(* CODESYS project Initial_Program_RECOVERED_2024-04-08T14-02-49.project
   Version: 0.0.0.0
   Title: Initial_Program
   Author: MYBOOK

Project tree, tasks and I/O mapping:
  Skripsi_Yosef : TM262L10MESE8T, Schneider Electric, order no. TM262L10MESE8T, version 5.0.4.83
      settings: Enable OPC-UA Server = True; BinaryFileSize = 968; Dhcps Host 0.Client Device Name = 'DEVICE_1'; Dhcps Host 0.Client IP Address = [192, 168, 3, 3]; Dhcps Host 0.Network Mask = [255, 255, 255, 0]; Dhcps Host 0.Default Gateway = [192, 168, 3, 254]; serialized Values = 512f82cd-0d03-416a-ab18-865b7c93dff8=0|; InterfaceUsedByDhcpSize = 4; InterfaceUsedByDhcp = [192,168,3,254]
    application Application
      task MAST (cyclic, interval 10 ms, priority 15, watchdog 50 ms x 1) calls SR_Main
      program SR_Main [LD]
      global variables GVL
    Machine Assistant
    Message Logger
    Ethernet_1 : ETH1, Schneider Electric, version 5.0.4.83
        settings: DeviceName = 'M262'; WebServer = FALSE; FTP Server = TRUE; SoMachine Protocol = FALSE; Modbus Server = FALSE; NetManage Protocol = FALSE; SNMP protocol = FALSE; WebVisu protocol = FALSE; DHCP Server Active = TRUE; Secured Web Server = TRUE; Remote Connection = FALSE
    IO_Bus : IO bus - TM3, Schneider Electric, version 5.0.4.83
    DI : Digital Inputs, Schneider Electric, version 5.0.4.83
        input  ibDI_IB0 : BYTE  // IB0
        input  ibDI_IB1 : BYTE  // IB1
    COM_Bus : COM Bus - TMS, Schneider Electric, version 5.0.4.83
    DQ : Digital Outputs, Schneider Electric, version 5.0.4.83
        output qbDQ_QB0 : BYTE  // QB0
        output qbDQ_QB1 : BYTE  // QB1
    Ethernet_2 : ETH2, Schneider Electric, version 5.0.4.83
        settings: IPAddress = [192, 168, 3, 254]; SubnetMask = [255, 255, 255, 0]; GatewayAddress = [192, 168, 3, 1]; DeviceName = 'M262_PLC'; WebServer = TRUE; FTP Server = TRUE; SoMachine Protocol = TRUE; Modbus Server = TRUE; NetManage Protocol = TRUE; SNMP protocol = TRUE; WebVisu protocol = FALSE; DHCP Server Active = TRUE; Secured Web Server = TRUE; Remote Connection = TRUE
      Modbus_TCP_IO_Scanner : Modbus TCP IO Scanner, Schneider Electric, version 1.0.0.12
          unmapped channels: Global Status, Healthbit 0, Healthbit 1, Healthbit 2, Healthbit 3
        Generic_Modbus_TCP_Slave : Generic Modbus TCP Slave, Schneider Electric, version 1.0.2.21
            settings: DeviceNumber = 512; Object Input1 = [128, 1, 21233765, 0]; Unit-ID = 248; IPAddress = [192, 168, 3, 3]; GatewayAddress = [192, 168, 3, 254]; DeviceName = 'DEVICE_1'; AC_Temp.Channel ID = 0; AC_Temp.Unit-ID = 255; AC_Temp.Repetition Rate = 20; AC_Temp.Function Code = 3; AC_Temp.Read Offset = 16#0065; AC_Temp.Read Length = 1; AC_Temp.Write Offset = 0; AC_Temp.Write Length = 0
            unmapped channels: AC_Temp
    Serial_Line : Serial line, Schneider Electric, version 5.0.4.83
      Machine_Expert_Network_Manager : Machine Expert-Network Manager, Schneider Electric, version 4.0.0.3 (disabled)
  Project Information/
    function GetVersion [ST]
    function GetCompany [ST]
    function GetTitle [ST]
    function GetTextProperty2 [ST]
    function GetTextProperty [ST]
    function GetBooleanProperty [ST]
    function GetVersionProperty [ST]
    function GetNumberProperty [ST]
*)

// Skripsi_Yosef/Application/GVL
{attribute 'qualified_only'}
VAR_GLOBAL
END_VAR

// Skripsi_Yosef/Application/SR_Main
PROGRAM SR_Main
VAR
END_VAR

// NETWORK 1

END_PROGRAM

// Project Information/GetVersion
// This function has been automatically generated from the project information.
{attribute 'signature_flag' := '1073741824'}
{attribute 'register_in_runtime'}
FUNCTION GetVersion : VERSION
VAR_INPUT
	
END_VAR

GetVersion.uiMajor := 0;
GetVersion.uiMinor := 0;
GetVersion.uiServicePack := 0;
GetVersion.uiPatch := 0;

END_FUNCTION

// Project Information/GetCompany
// This function has been automatically generated from the project information.
{attribute 'signature_flag' := '1073741824'}
{attribute 'register_in_runtime'}
FUNCTION GetCompany : WSTRING
VAR_INPUT
	
END_VAR

GetCompany := "";

END_FUNCTION

// Project Information/GetTitle
// This function has been automatically generated from the project information.
{attribute 'signature_flag' := '1073741824'}
{attribute 'register_in_runtime'}
FUNCTION GetTitle : WSTRING
VAR_INPUT
	
END_VAR

GetTitle := "Initial_Program";

END_FUNCTION

// Project Information/GetTextProperty2
// This function has been automatically generated from the project information.
{attribute 'signature_flag' := '1073741824'}
{attribute 'register_in_runtime'}
FUNCTION GetTextProperty2 : POINTER TO WSTRING
VAR_INPUT
	stKey: WSTRING;
END_VAR

IF stKey = "Author" THEN
	GetTextProperty2 := ADR("MYBOOK");
ELSIF stKey = "Company" THEN
	GetTextProperty2 := ADR("");
ELSIF stKey = "Description" THEN
	GetTextProperty2 := ADR("");
ELSIF stKey = "Project" THEN
	GetTextProperty2 := ADR("Initial_Program");
ELSIF stKey = "Title" THEN
	GetTextProperty2 := ADR("Initial_Program");
ELSE
	GetTextProperty2 := ADR("");
END_IF

END_FUNCTION

// Project Information/GetTextProperty
// This function has been automatically generated from the project information.
{attribute 'signature_flag' := '1073741824'}
{attribute 'register_in_runtime'}
FUNCTION GetTextProperty : WSTRING
VAR_INPUT
	stKey: WSTRING;
END_VAR

IF stKey = "Author" THEN
	GetTextProperty := "MYBOOK";
ELSIF stKey = "Company" THEN
	GetTextProperty := "";
ELSIF stKey = "Description" THEN
	GetTextProperty := "";
ELSIF stKey = "Project" THEN
	GetTextProperty := "Initial_Program";
ELSIF stKey = "Title" THEN
	GetTextProperty := "Initial_Program";
ELSE
	GetTextProperty := "";
END_IF

END_FUNCTION

// Project Information/GetBooleanProperty
// This function has been automatically generated from the project information.
{attribute 'signature_flag' := '1073741824'}
{attribute 'register_in_runtime'}
FUNCTION GetBooleanProperty : BOOL
VAR_INPUT
	stKey: WSTRING;
END_VAR

GetBooleanProperty := FALSE;

END_FUNCTION

// Project Information/GetVersionProperty
// This function has been automatically generated from the project information.
{attribute 'signature_flag' := '1073741824'}
{attribute 'register_in_runtime'}
FUNCTION GetVersionProperty : VERSION
VAR_INPUT
	stKey: WSTRING;
END_VAR

IF stKey = "Version" THEN
	GetVersionProperty.uiMajor := 0;
	GetVersionProperty.uiMinor := 0;
	GetVersionProperty.uiServicePack := 0;
	GetVersionProperty.uiPatch := 0;
ELSE
	GetVersionProperty.uiMajor := 0;
	GetVersionProperty.uiMinor := 0;
	GetVersionProperty.uiServicePack := 0;
	GetVersionProperty.uiPatch := 0;
END_IF

END_FUNCTION

// Project Information/GetNumberProperty
// This function has been automatically generated from the project information.
{attribute 'signature_flag' := '1073741824'}
{attribute 'register_in_runtime'}
FUNCTION GetNumberProperty : DINT
VAR_INPUT
	stKey: WSTRING;
END_VAR

GetNumberProperty := 0;

END_FUNCTION
